(* IEC 61131-3 sources: pandora/pandora/aws-platform-main/aws-platform-main/src/Hmi/Modules, 5 files *)

(* ---- IJoystick.st ---- *)
NAMESPACE Esab.Hmi.Modules

    INTERFACE IJoystick
        /// Cyclic execute
        METHOD Execute
        END_METHOD

        /// Returns the current direction (position) of the joystick
        METHOD GetPosition : JoystickPosition
        END_METHOD

        /// Sets the click listener
        METHOD SetClickListener
            VAR_INPUT
                listener : IClickListener;
            END_VAR
        END_METHOD

        /// Sets the long hold listener
        METHOD SetLongHoldListener
            VAR_INPUT
                listener : ILongHoldListener;
            END_VAR
        END_METHOD

        /// Sets the position changed listener
        METHOD SetPositionChangedListener
            VAR_INPUT
                listener : IPositionChangedListener;
            END_VAR
        END_METHOD
    END_INTERFACE

    INTERFACE IClickListener
        /// Called when the joystick is clicked
        METHOD OnClick
            VAR_INPUT
                direction : JoystickPosition;
            END_VAR
        END_METHOD
    END_INTERFACE

    INTERFACE ILongHoldListener
        /// Called when long hold is first detected
        METHOD OnLongHoldDetected
            VAR_INPUT
                direction : JoystickPosition;
            END_VAR
        END_METHOD

        /// Called every execution cycle until release
        METHOD OnLongHold
            VAR_INPUT
                direction : JoystickPosition;
            END_VAR
        END_METHOD

        /// Called when the joystick is released after a long hold
        /// The direction will be the direction the joystick was held in before release
        METHOD OnLongHoldReleased
            VAR_INPUT
                direction : JoystickPosition;
            END_VAR
        END_METHOD
    END_INTERFACE

    INTERFACE IPositionChangedListener
        /// Called when the joysticks direction changes
        METHOD OnPositionChanged
            VAR_INPUT
                position : JoystickPosition;
            END_VAR
        END_METHOD
    END_INTERFACE

    TYPE
        JoystickPosition : INT(None := -1,
                               Center := 0,
                               Up := 1,
                               Down := 2,
                               Triangle := 3,
                               Square := 4
                           ) := Center;
    END_TYPE

END_NAMESPACE

(* ---- PushButton.st ---- *)
USING Esab.Utils.Alarming;
USING Esab.Utils.Assets;
USING Esab.Utils.Timer;
USING Esab.Io;

NAMESPACE Esab.Hmi.Modules

    CLASS PushButton EXTENDS Asset IMPLEMENTS IPushButton
        VAR PRIVATE
            _io : REF_TO PushButtonIo;
            _onTimer : ITimer;
            _listener : IPushButtonListener := NULL;

            _status : BOOL := FALSE;
            _shadowStatus : BOOL := FALSE;
            _statusFrequency : LREAL := 0.0;
        END_VAR

        METHOD PUBLIC Setup
            VAR_INPUT
                io : REF_TO PushButtonIo;
                onTimer : ITimer := NULL;
                setupAlarm : IAlarm;
            END_VAR

            _io := io;
            _onTimer := onTimer;
            _setupAlarm := setupAlarm;

            _isSetup := _io <> NULL;
        END_METHOD

        METHOD PUBLIC OVERRIDE Execute
            SUPER.Execute();

            IF _setupAlarm.IsActive() THEN
                RETURN;
            END_IF;

            IF _listener <> NULL THEN
                IF _io^.Pressed.RisingEdge() THEN
                    _listener.OnPushButtonPressed(THIS.GetIdentifier());
                ELSIF _io^.Pressed.GetValue() THEN
                    _listener.OnPushButton(THIS.GetIdentifier());
                ELSIF _io^.Pressed.FallingEdge() THEN
                    _listener.OnPushButtonReleased(THIS.GetIdentifier());
                END_IF;
            END_IF;

            THIS.UpdateStatus();
        END_METHOD

        METHOD PUBLIC OVERRIDE Observe : IAssetObservable
            Observe := NULL; // Push button cannot be observed
        END_METHOD

        METHOD PUBLIC IsPressed : BOOL
            IsPressed := _io^.Pressed.GetValue();
        END_METHOD

        METHOD PUBLIC SetStatus
            VAR_INPUT
                status : BOOL := FALSE;
            END_VAR

            _status := status;
            _shadowStatus := _status;
            _statusFrequency := 0.0;

            THIS.UpdateStatus();
        END_METHOD

        METHOD PUBLIC SetStatus
            VAR_INPUT
                frequency : LREAL := 0.0;
            END_VAR

            _status := TRUE;
            _shadowStatus := _status;
            _statusFrequency := frequency;

            THIS.UpdateStatus();
        END_METHOD

        METHOD PUBLIC SetListener
            VAR_INPUT
                listener : IPushButtonListener;
            END_VAR

            _listener := listener;
        END_METHOD

        METHOD PRIVATE UpdateStatus
            IF _status THEN
                IF _onTimer <> NULL AND _statusFrequency > 0.1 THEN
                    _onTimer.Execute(TRUE, TO_LTIME(TO_LINT((1.0/_statusFrequency)/2.0*1000.0)));
                    IF _onTimer.Expired() THEN
                        _onTimer.Execute(FALSE);
                        _shadowStatus := NOT _shadowStatus;
                    END_IF;
                ELSE
                    _shadowStatus := _status;
                END_IF;
            ELSE
                IF _onTimer <> NULL THEN
                    _onTimer.Execute(FALSE);
                END_IF;

                _shadowStatus := FALSE;
            END_IF;

            _io^.Status.SetValue(_shadowStatus);
        END_METHOD
    END_CLASS

    TYPE
        PushButtonIo : STRUCT
            Pressed : DigitalInput;
            Status : DigitalOutput;
        END_STRUCT;
    END_TYPE

END_NAMESPACE

(* ---- TwinPushButton.st ---- *)
USING Esab.Utils.Alarming;
USING Esab.Utils.Assets;
USING Esab.Io;

NAMESPACE Esab.Hmi.Modules

    CLASS TwinPushButton EXTENDS Asset IMPLEMENTS ITwinPushButton
        VAR PRIVATE
            _io : REF_TO TwinPushButtonIo;
            _listener : IPushButtonListener := NULL;
        END_VAR

        METHOD PUBLIC Setup
            VAR_INPUT
                io : REF_TO TwinPushButtonIo;
                setupAlarm : IAlarm;
            END_VAR

            _io := io;
            _setupAlarm := setupAlarm;

            _isSetup := _io <> NULL;
        END_METHOD

        METHOD PUBLIC OVERRIDE Observe : IAssetObservable
            Observe := NULL; // Push button cannot be observed
        END_METHOD

        METHOD PUBLIC OVERRIDE Execute
            SUPER.Execute();

            IF _setupAlarm.IsActive() THEN
                RETURN;
            END_IF;

            IF _listener <> NULL THEN
                IF _io^.Direction1.RisingEdge() OR _io^.Direction2.RisingEdge() THEN
                    _listener.OnPushButtonPressed(THIS.GetIdentifier());
                ELSIF _io^.Direction1.GetValue() OR _io^.Direction2.GetValue() THEN
                    _listener.OnPushButton(THIS.GetIdentifier());
                ELSIF _io^.Direction1.FallingEdge() OR _io^.Direction2.FallingEdge() THEN
                    _listener.OnPushButtonReleased(THIS.GetIdentifier());
                END_IF;
            END_IF;
        END_METHOD

        METHOD PUBLIC IsPressed : BOOL
            IsPressed := THIS.IsInDirection1() OR THIS.IsInDirection2();
        END_METHOD

        METHOD PUBLIC IsInDirection1 : BOOL
            IsInDirection1 := _io^.Direction1.GetValue();
        END_METHOD

        METHOD PUBLIC IsInDirection2 : BOOL
            IsInDirection2 := _io^.Direction2.GetValue();
        END_METHOD

        METHOD PUBLIC SetStatus
            VAR_INPUT
                status : BOOL := FALSE;
            END_VAR

            _io^.Status.SetValue(status);
        END_METHOD

        METHOD PUBLIC SetStatus
            VAR_INPUT
                frequency : LREAL := 0.0;
            END_VAR

            ;
        END_METHOD

        METHOD PUBLIC SetListener
            VAR_INPUT
                listener : IPushButtonListener;
            END_VAR

            _listener := listener;
        END_METHOD
    END_CLASS

    TYPE
        TwinPushButtonIo : STRUCT
            Direction1 : DigitalInput;
            Direction2 : DigitalInput;
            Status : DigitalOutput;
        END_STRUCT;
    END_TYPE

END_NAMESPACE

(* ---- IPushButton.st ---- *)
NAMESPACE Esab.Hmi.Modules

    INTERFACE IPushButton
        METHOD IsPressed : BOOL
        END_METHOD

        METHOD SetStatus
            VAR_INPUT
                status : BOOL := FALSE;
            END_VAR
        END_METHOD

        METHOD SetStatus
            VAR_INPUT
                frequency : LREAL := 0.0;
            END_VAR
        END_METHOD

        METHOD SetListener
            VAR_INPUT
                listener : IPushButtonListener;
            END_VAR
        END_METHOD
    END_INTERFACE

    INTERFACE ITwinPushButton EXTENDS IPushButton
        METHOD IsInDirection1 : BOOL
        END_METHOD

        METHOD IsInDirection2 : BOOL
        END_METHOD
    END_INTERFACE

    INTERFACE IPushButtonListener
        METHOD OnPushButtonPressed
            VAR_INPUT
                id : Esab.AssetIdentifier;
            END_VAR
        END_METHOD

        METHOD OnPushButton
            VAR_INPUT
                id : Esab.AssetIdentifier;
            END_VAR
        END_METHOD

        METHOD OnPushButtonReleased
            VAR_INPUT
                id : Esab.AssetIdentifier;
            END_VAR
        END_METHOD
    END_INTERFACE

END_NAMESPACE

(* ---- DiscreteJoystick.st ---- *)
USING Esab.Io;
USING Esab.Utils.Alarming;
USING Esab.Utils.Assets;
USING Esab.Utils.Timer;
USING Esab.Hmi.Modules;

USING Siemens.Simatic.S71500.Alarming;

NAMESPACE Esab.Hmi.Modules

    CLASS DiscreteJoystick EXTENDS Asset IMPLEMENTS IJoystick
        VAR PUBLIC
        END_VAR

        VAR PRIVATE
            _io : REF_TO DiscreteJoystickIo;
            _longHoldTimer : ITimer := NULL;

            _previousPosition : JoystickPosition := JoystickPosition#Center;
            _placementChangedDirection : JoystickPosition := JoystickPosition#None;
            _lastLongHold : BOOL := FALSE;
            _longHold : BOOL;

            _clickListener : IClickListener;
            _longHoldListener : ILongHoldListener;
            _directionListener : IPositionChangedListener;
        END_VAR

        METHOD PUBLIC Setup
            VAR_INPUT
                io : REF_TO DiscreteJoystickIo;
                longHoldTimer : ITimer;
                setupAlarm : IAlarm;
            END_VAR

            _io := io;
            _longHoldTimer := longHoldTimer;
            _setupAlarm := setupAlarm;

            _isSetup := _io <> NULL AND _longHoldTimer <> NULL;
        END_METHOD

        METHOD PUBLIC OVERRIDE Execute
            VAR_TEMP
                _newPosition : JoystickPosition;
            END_VAR

            SUPER.Execute();

            IF _setupAlarm.IsActive() THEN
                RETURN;
            END_IF;

            _newPosition := THIS.GetPosition();

            IF _longHoldListener <> NULL THEN
                _longHoldTimer.Execute(_io^.Up.GetValue() OR _io^.Down.GetValue() OR _io^.Triangle.GetValue() OR _io^.Square.GetValue(), LT#1s);
                _longHold := _longHoldTimer.Expired();

                IF _longHold AND NOT _lastLongHold THEN
                    _longHoldListener.OnLongHoldDetected(THIS.GetPosition());
                ELSIF _longHold AND _lastLongHold THEN
                    _longHoldListener.OnLongHold(THIS.GetPosition());
                ELSIF NOT _longHold AND _lastLongHold THEN
                    _longHoldListener.OnLongHoldReleased(_previousPosition);
                END_IF;
            ELSE
                _longHoldTimer.Execute(FALSE, LT#1s);
                _longHold := FALSE;
            END_IF;

            IF _clickListener <> NULL THEN
                IF _newPosition = JoystickPosition#Center &&
                   _previousPosition <> JoystickPosition#Center &&
                    NOT (_longHold OR _lastLongHold) THEN

                    _clickListener.OnClick(_previousPosition);
                END_IF;
            END_IF;

            IF _directionListener <> NULL THEN
                IF _newPosition <> _previousPosition THEN
                    _directionListener.OnPositionChanged(_newPosition);
                END_IF;
            END_IF;

            _lastLongHold := _longHold;
            _previousPosition := _newPosition;
        END_METHOD

        METHOD PUBLIC GetPosition : JoystickPosition
            IF NOT _isSetup THEN
                RETURN;
            END_IF;

            IF _io^.Up.GetValue() THEN
                GetPosition := JoystickPosition#Up;
            ELSIF _io^.Down.GetValue() THEN
                GetPosition := JoystickPosition#Down;
            ELSIF _io^.Triangle.GetValue() THEN
                GetPosition := JoystickPosition#Triangle;
            ELSIF _io^.Square.GetValue() THEN
                GetPosition := JoystickPosition#Square;
            ELSE
                GetPosition := JoystickPosition#Center;
            END_IF;
        END_METHOD

        METHOD PUBLIC SetClickListener
            VAR_INPUT
                listener : IClickListener;
            END_VAR

            _clickListener := listener;
        END_METHOD

        METHOD PUBLIC SetLongHoldListener
            VAR_INPUT
                listener : ILongHoldListener;
            END_VAR

            _longHoldListener := listener;
        END_METHOD

        METHOD PUBLIC SetPositionChangedListener
            VAR_INPUT
                listener : IPositionChangedListener;
            END_VAR

            _directionListener := listener;
        END_METHOD

        METHOD PUBLIC OVERRIDE Observe : IAssetObservable
            Observe := NULL; // Joystick does not currently have an observable.
        END_METHOD
    END_CLASS

    TYPE
        DiscreteJoystickIo : STRUCT
            Up : DigitalInput;
            Down : DigitalInput;
            Triangle : DigitalInput;
            Square : DigitalInput;
        END_STRUCT;
    END_TYPE

END_NAMESPACE
